  MoveL 11286 to (240.02, 46.51, 153.89) mm, rotated rx 180 ry 0 rz 180 deg; joints [-155.698, -65.543, -49.369, 46.991, 34.25, -41.545]
  MoveL 11287 to (240.02, 46.51, 153.89) mm, rotated rx 180 ry 0 rz 180 deg; joints [-155.698, -65.543, -49.369, 46.991, 34.25, -41.545]
  Call Extruder(208.81911)
  MoveL 11288 to (240.06, 46.72, 153.89) mm, rotated rx -180 ry 0 rz -180 deg; joints [-155.682, -65.561, -49.333, 47.032, 34.249, -41.586]
  MoveL 11289 to (240.06, 46.72, 153.89) mm, rotated rx -180 ry 0 rz -180 deg; joints [-155.682, -65.561, -49.333, 47.032, 34.249, -41.586]
  Call Extruder(208.93371)
  MoveL 11290 to (240.11, 46.92, 153.89) mm, rotated rx 180 ry 0 rz 180 deg; joints [-155.665, -65.578, -49.298, 47.072, 34.247, -41.627]
  MoveL 11291 to (240.11, 46.92, 153.89) mm, rotated rx 180 ry 0 rz 180 deg; joints [-155.665, -65.578, -49.298, 47.072, 34.247, -41.627]
  Call Extruder(209.04786)
  MoveL 11292 to (240.15, 47.12, 153.89) mm, rotated rx 180 ry 0 rz 180 deg; joints [-155.649, -65.596, -49.263, 47.113, 34.246, -41.668]
  MoveL 11293 to (240.15, 47.12, 153.89) mm, rotated rx 180 ry 0 rz 180 deg; joints [-155.649, -65.596, -49.263, 47.113, 34.246, -41.668]
  Call Extruder(209.16155)
  MoveL 11294 to (240.2, 47.33, 153.89) mm, rotated rx 180 ry 0 rz 180 deg; joints [-155.633, -65.614, -49.227, 47.154, 34.245, -41.71]
  MoveL 11295 to (240.2, 47.33, 153.89) mm, rotated rx 180 ry 0 rz 180 deg; joints [-155.633, -65.614, -49.227, 47.154, 34.245, -41.71]
  Call Extruder(209.28696)
  MoveL 11296 to (240.24, 47.55, 153.89) mm, rotated rx 180 ry 0 rz 180 deg; joints [-155.614, -65.633, -49.188, 47.199, 34.244, -41.755]
  MoveL 11297 to (240.24, 47.55, 153.89) mm, rotated rx 180 ry 0 rz 180 deg; joints [-155.614, -65.633, -49.188, 47.199, 34.244, -41.755]
  Call Extruder(209.42394)
  MoveL 11298 to (240.29, 47.8, 153.89) mm, rotated rx 180 ry 0 rz 180 deg; joints [-155.594, -65.654, -49.146, 47.249, 34.243, -41.804]
  MoveL 11299 to (240.29, 47.8, 153.89) mm, rotated rx 180 ry 0 rz 180 deg; joints [-155.594, -65.654, -49.146, 47.249, 34.243, -41.804]
  Call Extruder(209.56031)
  MoveL 11300 to (240.34, 48.05, 153.89) mm, rotated rx 180 ry 0 rz 180 deg; joints [-155.574, -65.675, -49.104, 47.298, 34.242, -41.854]
  MoveL 11301 to (240.34, 48.05, 153.89) mm, rotated rx 180 ry 0 rz 180 deg; joints [-155.574, -65.675, -49.104, 47.298, 34.242, -41.854]
  Call Extruder(209.69607)
  MoveL 11302 to (240.39, 48.3, 153.89) mm, rotated rx 180 ry 0 rz 180 deg; joints [-155.554, -65.696, -49.061, 47.348, 34.241, -41.904]
  MoveL 11303 to (240.39, 48.3, 153.89) mm, rotated rx 180 ry 0 rz 180 deg; joints [-155.554, -65.696, -49.061, 47.348, 34.241, -41.904]
  Call Extruder(209.83121)
  MoveL 11304 to (240.44, 48.55, 153.89) mm, rotated rx 180 ry 0 rz 180 deg; joints [-155.534, -65.717, -49.019, 47.398, 34.24, -41.954]
  MoveL 11305 to (240.44, 48.55, 153.89) mm, rotated rx 180 ry 0 rz 180 deg; joints [-155.534, -65.717, -49.019, 47.398, 34.24, -41.954]
  Call Extruder(209.96575)
  MoveL 11306 to (240.49, 48.8, 153.89) mm, rotated rx -180 ry 0 rz 180 deg; joints [-155.514, -65.738, -48.977, 47.447, 34.239, -42.003]
  MoveL 11307 to (240.49, 48.8, 153.89) mm, rotated rx -180 ry 0 rz 180 deg; joints [-155.514, -65.738, -48.977, 47.447, 34.239, -42.003]
  Call Extruder(210.09968)
  MoveL 11308 to (240.54, 49.05, 153.89) mm, rotated rx 180 ry 0 rz 180 deg; joints [-155.494, -65.759, -48.935, 47.497, 34.238, -42.053]
  MoveL 11309 to (240.54, 49.05, 153.89) mm, rotated rx 180 ry 0 rz 180 deg; joints [-155.494, -65.759, -48.935, 47.497, 34.238, -42.053]
  Call Extruder(210.24754)
  MoveL 11310 to (240.59, 49.33, 153.89) mm, rotated rx -180 ry 0 rz 180 deg; joints [-155.471, -65.782, -48.889, 47.551, 34.238, -42.108]
  MoveL 11311 to (240.59, 49.33, 153.89) mm, rotated rx -180 ry 0 rz 180 deg; joints [-155.471, -65.782, -48.889, 47.551, 34.238, -42.108]
  Call Extruder(210.40929)
  MoveL 11312 to (240.64, 49.63, 153.89) mm, rotated rx 180 ry 0 rz -180 deg; joints [-155.446, -65.806, -48.84, 47.611, 34.238, -42.167]
  MoveL 11313 to (240.64, 49.63, 153.89) mm, rotated rx 180 ry 0 rz -180 deg; joints [-155.446, -65.806, -48.84, 47.611, 34.238, -42.167]
  Call Extruder(210.57031)
  MoveL 11314 to (240.69, 49.94, 153.89) mm, rotated rx -180 ry 0 rz 180 deg; joints [-155.421, -65.831, -48.791, 47.671, 34.238, -42.227]
  MoveL 11315 to (240.69, 49.94, 153.89) mm, rotated rx -180 ry 0 rz 180 deg; joints [-155.421, -65.831, -48.791, 47.671, 34.238, -42.227]
  Call Extruder(210.73060)
  MoveL 11316 to (240.74, 50.24, 153.89) mm, rotated rx -180 ry 0 rz 180 deg; joints [-155.396, -65.855, -48.742, 47.73, 34.239, -42.287]
  MoveL 11317 to (240.74, 50.24, 153.89) mm, rotated rx -180 ry 0 rz 180 deg; joints [-155.396, -65.855, -48.742, 47.73, 34.239, -42.287]
  Call Extruder(210.89016)
  MoveL 11318 to (240.78, 50.55, 153.89) mm, rotated rx 180 ry 0 rz 180 deg; joints [-155.371, -65.88, -48.693, 47.79, 34.239, -42.346]
  MoveL 11319 to (240.78, 50.55, 153.89) mm, rotated rx 180 ry 0 rz 180 deg; joints [-155.371, -65.88, -48.693, 47.79, 34.239, -42.346]
  Call Extruder(211.04899)
  MoveL 11320 to (240.83, 50.86, 153.89) mm, rotated rx 180 ry 0 rz 180 deg; joints [-155.346, -65.904, -48.644, 47.85, 34.239, -42.406]
  MoveL 11321 to (240.83, 50.86, 153.89) mm, rotated rx 180 ry 0 rz 180 deg; joints [-155.346, -65.904, -48.644, 47.85, 34.239, -42.406]
  Call Extruder(211.22766)
  MoveL 11322 to (240.88, 51.2, 153.89) mm, rotated rx 180 ry 0 rz 180 deg; joints [-155.317, -65.931, -48.59, 47.917, 34.241, -42.473]
  MoveL 11323 to (240.88, 51.2, 153.89) mm, rotated rx 180 ry 0 rz 180 deg; joints [-155.317, -65.931, -48.59, 47.917, 34.241, -42.473]
  Call Extruder(211.42611)
  MoveL 11324 to (240.92, 51.59, 153.89) mm, rotated rx 180 ry 0 rz -180 deg; joints [-155.285, -65.96, -48.531, 47.991, 34.243, -42.546]
  MoveL 11325 to (240.92, 51.59, 153.89) mm, rotated rx 180 ry 0 rz -180 deg; joints [-155.285, -65.96, -48.531, 47.991, 34.243, -42.546]
  Call Extruder(211.62368)
  MoveL 11326 to (240.97, 51.98, 153.89) mm, rotated rx 180 ry 0 rz -180 deg; joints [-155.252, -65.989, -48.473, 48.066, 34.245, -42.62]
  MoveL 11327 to (240.97, 51.98, 153.89) mm, rotated rx 180 ry 0 rz -180 deg; joints [-155.252, -65.989, -48.473, 48.066, 34.245, -42.62]
  Call Extruder(211.82039)
  MoveL 11328 to (241.02, 52.36, 153.89) mm, rotated rx -180 ry 0 rz 180 deg; joints [-155.22, -66.019, -48.414, 48.14, 34.247, -42.694]
  MoveL 11329 to (241.02, 52.36, 153.89) mm, rotated rx -180 ry 0 rz 180 deg; joints [-155.22, -66.019, -48.414, 48.14, 34.247, -42.694]
  Call Extruder(212.01622)
  MoveL 11330 to (241.06, 52.75, 153.89) mm, rotated rx 180 ry 0 rz 180 deg; joints [-155.188, -66.048, -48.356, 48.214, 34.25, -42.768]
  MoveL 11331 to (241.06, 52.75, 153.89) mm, rotated rx 180 ry 0 rz 180 deg; joints [-155.188, -66.048, -48.356, 48.214, 34.25, -42.768]
  Call Extruder(212.31166)
  MoveL 11332 to (241.11, 53.34, 153.89) mm, rotated rx -180 ry 0 rz 180 deg; joints [-155.138, -66.09, -48.272, 48.326, 34.256, -42.877]
  MoveL 11333 to (241.11, 53.34, 153.89) mm, rotated rx -180 ry 0 rz 180 deg; joints [-155.138, -66.09, -48.272, 48.326, 34.256, -42.877]
  Call Extruder(212.60577)
  MoveL 11334 to (241.16, 53.93, 153.89) mm, rotated rx -180 ry 0 rz 180 deg; joints [-155.088, -66.131, -48.188, 48.437, 34.262, -42.987]
  MoveL 11335 to (241.16, 53.93, 153.89) mm, rotated rx -180 ry 0 rz 180 deg; joints [-155.088, -66.131, -48.188, 48.437, 34.262, -42.987]
  Call Extruder(212.89854)
  MoveL 11336 to (241.2, 54.52, 153.89) mm, rotated rx -180 ry 0 rz 180 deg; joints [-155.038, -66.173, -48.104, 48.548, 34.268, -43.096]
  MoveL 11337 to (241.2, 54.52, 153.89) mm, rotated rx -180 ry 0 rz 180 deg; joints [-155.038, -66.173, -48.104, 48.548, 34.268, -43.096]
  Call Extruder(213.47199)
  MoveL 11338 to (241.25, 55.68, 153.89) mm, rotated rx 180 ry 0 rz 180 deg; joints [-154.938, -66.25, -47.95, 48.763, 34.285, -43.307]
  MoveL 11339 to (241.25, 55.68, 153.89) mm, rotated rx 180 ry 0 rz 180 deg; joints [-154.938, -66.25, -47.95, 48.763, 34.285, -43.307]
  Call Extruder(214.18582)
  MoveL 11340 to (241.29, 57.14, 153.89) mm, rotated rx 180 ry 0 rz 180 deg; joints [-154.812, -66.345, -47.76, 49.03, 34.309, -43.568]
  Call Extruder(256.25069)
  MoveL 11341 to (241.29, 142.86, 153.89) mm, rotated rx -180 ry 0 rz 180 deg; joints [-147.778, -73.071, -34.392, 64.539, 36.196, -59.459]
  Call Extruder(256.67912)
  MoveL 11342 to (241.27, 143.73, 153.89) mm, rotated rx -180 ry 0 rz 180 deg; joints [-147.711, -73.155, -34.226, 64.698, 36.219, -59.631]
  MoveL 11343 to (241.27, 143.73, 153.89) mm, rotated rx -180 ry 0 rz 180 deg; joints [-147.711, -73.155, -34.226, 64.698, 36.219, -59.631]
  Call Extruder(257.25257)
  MoveL 11344 to (241.22, 144.9, 153.89) mm, rotated rx 180 ry 0 rz 180 deg; joints [-147.62, -73.265, -34.01, 64.907, 36.253, -59.856]
  MoveL 11345 to (241.22, 144.9, 153.89) mm, rotated rx 180 ry 0 rz 180 deg; joints [-147.62, -73.265, -34.01, 64.907, 36.253, -59.856]
  Call Extruder(257.68690)
  MoveL 11346 to (241.18, 145.77, 153.89) mm, rotated rx 180 ry 0 rz 180 deg; joints [-147.551, -73.346, -33.851, 65.062, 36.279, -60.024]
  MoveL 11347 to (241.18, 145.77, 153.89) mm, rotated rx 180 ry 0 rz 180 deg; joints [-147.551, -73.346, -33.851, 65.062, 36.279, -60.024]
  Call Extruder(257.98101)
  MoveL 11348 to (241.13, 146.36, 153.89) mm, rotated rx 180 ry 0 rz -180 deg; joints [-147.504, -73.398, -33.748, 65.165, 36.299, -60.133]
  MoveL 11349 to (241.13, 146.36, 153.89) mm, rotated rx 180 ry 0 rz -180 deg; joints [-147.504, -73.398, -33.748, 65.165, 36.299, -60.133]
  Call Extruder(258.27645)
  MoveL 11350 to (241.09, 146.95, 153.89) mm, rotated rx 180 ry 0 rz 180 deg; joints [-147.457, -73.451, -33.644, 65.267, 36.318, -60.243]
  MoveL 11351 to (241.09, 146.95, 153.89) mm, rotated rx 180 ry 0 rz 180 deg; joints [-147.457, -73.451, -33.644, 65.267, 36.318, -60.243]
  Call Extruder(258.52270)
  MoveL 11352 to (241.04, 147.44, 153.89) mm, rotated rx -180 ry 0 rz 180 deg; joints [-147.417, -73.493, -33.561, 65.351, 36.335, -60.333]
  MoveL 11353 to (241.04, 147.44, 153.89) mm, rotated rx -180 ry 0 rz 180 deg; joints [-147.417, -73.493, -33.561, 65.351, 36.335, -60.333]
  Call Extruder(258.71941)
  MoveL 11354 to (240.99, 147.83, 153.89) mm, rotated rx 180 ry 0 rz -180 deg; joints [-147.386, -73.525, -33.497, 65.416, 36.35, -60.402]
  MoveL 11355 to (240.99, 147.83, 153.89) mm, rotated rx 180 ry 0 rz -180 deg; joints [-147.386, -73.525, -33.497, 65.416, 36.35, -60.402]
  Call Extruder(258.91698)
  MoveL 11356 to (240.95, 148.22, 153.89) mm, rotated rx -180 ry 0 rz 180 deg; joints [-147.354, -73.557, -33.434, 65.481, 36.364, -60.471]
  MoveL 11357 to (240.95, 148.22, 153.89) mm, rotated rx -180 ry 0 rz 180 deg; joints [-147.354, -73.557, -33.434, 65.481, 36.364, -60.471]
  Call Extruder(259.11542)
  MoveL 11358 to (240.9, 148.6, 153.89) mm, rotated rx 180 ry 0 rz -180 deg; joints [-147.322, -73.59, -33.37, 65.546, 36.379, -60.541]
  MoveL 11359 to (240.9, 148.6, 153.89) mm, rotated rx 180 ry 0 rz -180 deg; joints [-147.322, -73.59, -33.37, 65.546, 36.379, -60.541]
  Call Extruder(259.31473)
  MoveL 11360 to (240.86, 148.99, 153.89) mm, rotated rx 180 ry 0 rz 180 deg; joints [-147.291, -73.622, -33.306, 65.611, 36.393, -60.61]
  MoveL 11361 to (240.86, 148.99, 153.89) mm, rotated rx 180 ry 0 rz 180 deg; joints [-147.291, -73.622, -33.306, 65.611, 36.393, -60.61]
  Call Extruder(259.47356)
  MoveL 11362 to (240.81, 149.3, 153.89) mm, rotated rx 180 ry 0 rz 180 deg; joints [-147.265, -73.646, -33.259, 65.661, 36.406, -60.663]
  MoveL 11363 to (240.81, 149.3, 153.89) mm, rotated rx 180 ry 0 rz 180 deg; joints [-147.265, -73.646, -33.259, 65.661, 36.406, -60.663]
  Call Extruder(259.63312)
  MoveL 11364 to (240.76, 149.6, 153.89) mm, rotated rx 180 ry 0 rz 180 deg; joints [-147.24, -73.67, -33.212, 65.71, 36.419, -60.715]
  MoveL 11365 to (240.76, 149.6, 153.89) mm, rotated rx 180 ry 0 rz 180 deg; joints [-147.24, -73.67, -33.212, 65.71, 36.419, -60.715]
  Call Extruder(259.79341)
  MoveL 11366 to (240.71, 149.91, 153.89) mm, rotated rx -180 ry 0 rz 180 deg; joints [-147.214, -73.694, -33.165, 65.76, 36.431, -60.767]
  MoveL 11367 to (240.71, 149.91, 153.89) mm, rotated rx -180 ry 0 rz 180 deg; joints [-147.214, -73.694, -33.165, 65.76, 36.431, -60.767]
  Call Extruder(259.95443)
  MoveL 11368 to (240.66, 150.21, 153.89) mm, rotated rx 180 ry 0 rz 180 deg; joints [-147.189, -73.718, -33.118, 65.809, 36.444, -60.819]
  MoveL 11369 to (240.66, 150.21, 153.89) mm, rotated rx 180 ry 0 rz 180 deg; joints [-147.189, -73.718, -33.118, 65.809, 36.444, -60.819]
  Call Extruder(260.11618)
  MoveL 11370 to (240.61, 150.52, 153.89) mm, rotated rx -180 ry 0 rz 180 deg; joints [-147.163, -73.742, -33.071, 65.859, 36.457, -60.872]
  MoveL 11371 to (240.61, 150.52, 153.89) mm, rotated rx -180 ry 0 rz 180 deg; joints [-147.163, -73.742, -33.071, 65.859, 36.457, -60.872]
  Call Extruder(260.27865)
  MoveL 11372 to (240.56, 150.83, 153.89) mm, rotated rx 180 ry 0 rz -180 deg; joints [-147.138, -73.765, -33.024, 65.908, 36.47, -60.924]
  MoveL 11373 to (240.56, 150.83, 153.89) mm, rotated rx 180 ry 0 rz -180 deg; joints [-147.138, -73.765, -33.024, 65.908, 36.47, -60.924]
  Call Extruder(260.41257)
  MoveL 11374 to (240.52, 151.07, 153.89) mm, rotated rx 180 ry 0 rz 180 deg; joints [-147.117, -73.784, -32.988, 65.947, 36.481, -60.965]
  MoveL 11375 to (240.52, 151.07, 153.89) mm, rotated rx 180 ry 0 rz 180 deg; joints [-147.117, -73.784, -32.988, 65.947, 36.481, -60.965]
  Call Extruder(260.54711)
  MoveL 11376 to (240.47, 151.32, 153.89) mm, rotated rx 180 ry 0 rz -180 deg; joints [-147.095, -73.801, -32.953, 65.986, 36.493, -61.006]
  MoveL 11377 to (240.47, 151.32, 153.89) mm, rotated rx 180 ry 0 rz -180 deg; joints [-147.095, -73.801, -32.953, 65.986, 36.493, -61.006]
  Call Extruder(260.68226)
  MoveL 11378 to (240.42, 151.57, 153.89) mm, rotated rx -180 ry 0 rz -180 deg; joints [-147.074, -73.819, -32.918, 66.025, 36.504, -61.046]
  MoveL 11379 to (240.42, 151.57, 153.89) mm, rotated rx -180 ry 0 rz -180 deg; joints [-147.074, -73.819, -32.918, 66.025, 36.504, -61.046]
  Call Extruder(260.81801)
  MoveL 11380 to (240.37, 151.82, 153.89) mm, rotated rx 180 ry 0 rz -180 deg; joints [-147.053, -73.837, -32.882, 66.064, 36.515, -61.087]
  MoveL 11381 to (240.37, 151.82, 153.89) mm, rotated rx 180 ry 0 rz -180 deg; joints [-147.053, -73.837, -32.882, 66.064, 36.515, -61.087]
  Call Extruder(260.95438)
  MoveL 11382 to (240.32, 152.07, 153.89) mm, rotated rx 180 ry 0 rz 180 deg; joints [-147.032, -73.855, -32.847, 66.102, 36.527, -61.128]
  MoveL 11383 to (240.32, 152.07, 153.89) mm, rotated rx 180 ry 0 rz 180 deg; joints [-147.032, -73.855, -32.847, 66.102, 36.527, -61.128]
  Call Extruder(261.09136)
  MoveL 11384 to (240.27, 152.32, 153.89) mm, rotated rx 180 ry 0 rz 180 deg; joints [-147.011, -73.874, -32.811, 66.141, 36.538, -61.169]
  MoveL 11385 to (240.27, 152.32, 153.89) mm, rotated rx 180 ry 0 rz 180 deg; joints [-147.011, -73.874, -32.811, 66.141, 36.538, -61.169]
  Call Extruder(261.22895)
  MoveL 11386 to (240.22, 152.57, 153.89) mm, rotated rx 180 ry 0 rz 180 deg; joints [-146.989, -73.892, -32.775, 66.18, 36.55, -61.209]
  MoveL 11387 to (240.22, 152.57, 153.89) mm, rotated rx 180 ry 0 rz 180 deg; joints [-146.989, -73.892, -32.775, 66.18, 36.55, -61.209]
  Call Extruder(261.34265)
  MoveL 11388 to (240.17, 152.77, 153.89) mm, rotated rx 180 ry 0 rz 180 deg; joints [-146.972, -73.906, -32.747, 66.211, 36.56, -61.242]
  MoveL 11389 to (240.17, 152.77, 153.89) mm, rotated rx 180 ry 0 rz 180 deg; joints [-146.972, -73.906, -32.747, 66.211, 36.56, -61.242]
  Call Extruder(261.45680)
  MoveL 11390 to (240.13, 152.98, 153.89) mm, rotated rx 180 ry 0 rz -180 deg; joints [-146.954, -73.92, -32.719, 66.242, 36.57, -61.275]
  MoveL 11391 to (240.13, 152.98, 153.89) mm, rotated rx 180 ry 0 rz -180 deg; joints [-146.954, -73.92, -32.719, 66.242, 36.57, -61.275]
  Call Extruder(261.57140)
  MoveL 11392 to (240.08, 153.18, 153.89) mm, rotated rx -180 ry 0 rz 180 deg; joints [-146.937, -73.935, -32.691, 66.274, 36.579, -61.307]
  MoveL 11393 to (240.08, 153.18, 153.89) mm, rotated rx -180 ry 0 rz 180 deg; joints [-146.937, -73.935, -32.691, 66.274, 36.579, -61.307]
  Call Extruder(261.68645)
  MoveL 11394 to (240.04, 153.39, 153.89) mm, rotated rx 180 ry 0 rz -180 deg; joints [-146.919, -73.949, -32.663, 66.305, 36.589, -61.34]
  MoveL 11395 to (240.04, 153.39, 153.89) mm, rotated rx 180 ry 0 rz -180 deg; joints [-146.919, -73.949, -32.663, 66.305, 36.589, -61.34]
  Call Extruder(261.80867)
  MoveL 11396 to (239.98, 153.6, 153.89) mm, rotated rx -180 ry 0 rz 180 deg; joints [-146.9, -73.962, -32.636, 66.336, 36.6, -61.372]
  MoveL 11397 to (239.98, 153.6, 153.89) mm, rotated rx -180 ry 0 rz 180 deg; joints [-146.9, -73.962, -32.636, 66.336, 36.6, -61.372]
  Call Extruder(261.93833)
  MoveL 11398 to (239.92, 153.82, 153.89) mm, rotated rx 180 ry 0 rz -180 deg; joints [-146.88, -73.975, -32.611, 66.367, 36.613, -61.404]
  MoveL 11399 to (239.92, 153.82, 153.89) mm, rotated rx 180 ry 0 rz -180 deg; joints [-146.88, -73.975, -32.611, 66.367, 36.613, -61.404]
  Call Extruder(262.06856)
  MoveL 11400 to (239.85, 154.05, 153.89) mm, rotated rx 180 ry 0 rz 180 deg; joints [-146.86, -73.988, -32.587, 66.399, 36.626, -61.435]
  MoveL 11401 to (239.85, 154.05, 153.89) mm, rotated rx 180 ry 0 rz 180 deg; joints [-146.86, -73.988, -32.587, 66.399, 36.626, -61.435]
  Call Extruder(262.19935)
  MoveL 11402 to (239.78, 154.27, 153.89) mm, rotated rx -180 ry 0 rz -180 deg; joints [-146.84, -74, -32.561, 66.43, 36.639, -61.467]
  MoveL 11403 to (239.78, 154.27, 153.89) mm, rotated rx -180 ry 0 rz -180 deg; joints [-146.84, -74, -32.561, 66.43, 36.639, -61.467]
  Call Extruder(262.33071)
  MoveL 11404 to (239.71, 154.49, 153.89) mm, rotated rx 180 ry 0 rz -180 deg; joints [-146.82, -74.013, -32.536, 66.461, 36.652, -61.499]
  MoveL 11405 to (239.71, 154.49, 153.89) mm, rotated rx 180 ry 0 rz -180 deg; joints [-146.82, -74.013, -32.536, 66.461, 36.652, -61.499]
  Call Extruder(262.44261)
  MoveL 11406 to (239.65, 154.68, 153.89) mm, rotated rx -180 ry 0 rz -180 deg; joints [-146.803, -74.023, -32.517, 66.487, 36.663, -61.525]
  MoveL 11407 to (239.65, 154.68, 153.89) mm, rotated rx -180 ry 0 rz -180 deg; joints [-146.803, -74.023, -32.517, 66.487, 36.663, -61.525]
  Call Extruder(262.55495)
  MoveL 11408 to (239.59, 154.87, 153.89) mm, rotated rx -180 ry 0 rz 180 deg; joints [-146.785, -74.033, -32.497, 66.513, 36.674, -61.551]
  MoveL 11409 to (239.59, 154.87, 153.89) mm, rotated rx -180 ry 0 rz 180 deg; joints [-146.785, -74.033, -32.497, 66.513, 36.674, -61.551]
  Call Extruder(262.66774)
  MoveL 11410 to (239.53, 155.06, 153.89) mm, rotated rx -180 ry 0 rz -180 deg; joints [-146.768, -74.043, -32.477, 66.538, 36.685, -61.577]
  MoveL 11411 to (239.53, 155.06, 153.89) mm, rotated rx -180 ry 0 rz -180 deg; joints [-146.768, -74.043, -32.477, 66.538, 36.685, -61.577]
  Call Extruder(262.78098)
  MoveL 11412 to (239.47, 155.25, 153.89) mm, rotated rx -180 ry 0 rz 180 deg; joints [-146.751, -74.054, -32.457, 66.564, 36.696, -61.603]
  MoveL 11413 to (239.47, 155.25, 153.89) mm, rotated rx -180 ry 0 rz 180 deg; joints [-146.751, -74.054, -32.457, 66.564, 36.696, -61.603]
  Call Extruder(262.89466)
  MoveL 11414 to (239.41, 155.44, 153.89) mm, rotated rx -180 ry 0 rz 180 deg; joints [-146.734, -74.064, -32.437, 66.59, 36.708, -61.629]
  MoveL 11415 to (239.41, 155.44, 153.89) mm, rotated rx -180 ry 0 rz 180 deg; joints [-146.734, -74.064, -32.437, 66.59, 36.708, -61.629]
  Call Extruder(263.07662)
  MoveL 11416 to (239.29, 155.73, 153.89) mm, rotated rx 180 ry 0 rz -180 deg; joints [-146.706, -74.075, -32.415, 66.626, 36.728, -61.664]
  MoveL 11417 to (239.29, 155.73, 153.89) mm, rotated rx 180 ry 0 rz -180 deg; joints [-146.706, -74.075, -32.415, 66.626, 36.728, -61.664]
  Call Extruder(263.25933)
  MoveL 11418 to (239.16, 156.02, 153.89) mm, rotated rx 180 ry 0 rz -180 deg; joints [-146.678, -74.087, -32.392, 66.661, 36.748, -61.699]
  MoveL 11419 to (239.16, 156.02, 153.89) mm, rotated rx 180 ry 0 rz -180 deg; joints [-146.678, -74.087, -32.392, 66.661, 36.748, -61.699]
  Call Extruder(263.42975)
  MoveL 11420 to (239.05, 156.29, 153.89) mm, rotated rx 180 ry 0 rz -180 deg; joints [-146.652, -74.097, -32.372, 66.694, 36.767, -61.73]
  MoveL 11421 to (239.05, 156.29, 153.89) mm, rotated rx 180 ry 0 rz -180 deg; joints [-146.652, -74.097, -32.372, 66.694, 36.767, -61.73]
  Call Extruder(263.58776)
  MoveL 11422 to (238.94, 156.54, 153.89) mm, rotated rx -180 ry 0 rz 180 deg; joints [-146.628, -74.106, -32.353, 66.724, 36.784, -61.759]
  MoveL 11423 to (238.94, 156.54, 153.89) mm, rotated rx -180 ry 0 rz 180 deg; joints [-146.628, -74.106, -32.353, 66.724, 36.784, -61.759]
  Call Extruder(263.74638)
  MoveL 11424 to (238.84, 156.79, 153.89) mm, rotated rx -180 ry 0 rz 180 deg; joints [-146.604, -74.116, -32.335, 66.754, 36.802, -61.788]
  MoveL 11425 to (238.84, 156.79, 153.89) mm, rotated rx -180 ry 0 rz 180 deg; joints [-146.604, -74.116, -32.335, 66.754, 36.802, -61.788]
  Call Extruder(263.95255)
  MoveL 11426 to (238.66, 157.09, 153.89) mm, rotated rx 180 ry 0 rz 180 deg; joints [-146.573, -74.12, -32.327, 66.784, 36.828, -61.814]
  MoveL 11427 to (238.66, 157.09, 153.89) mm, rotated rx 180 ry 0 rz 180 deg; joints [-146.573, -74.12, -32.327, 66.784, 36.828, -61.814]
  Call Extruder(264.15949)
  MoveL 11428 to (238.49, 157.4, 153.89) mm, rotated rx 180 ry 0 rz 180 deg; joints [-146.542, -74.124, -32.319, 66.813, 36.854, -61.84]
  MoveL 11429 to (238.49, 157.4, 153.89) mm, rotated rx 180 ry 0 rz 180 deg; joints [-146.542, -74.124, -32.319, 66.813, 36.854, -61.84]
  Call Extruder(264.36722)
  MoveL 11430 to (238.31, 157.7, 153.89) mm, rotated rx 180 ry 0 rz -180 deg; joints [-146.51, -74.128, -32.31, 66.843, 36.88, -61.866]
  MoveL 11431 to (238.31, 157.7, 153.89) mm, rotated rx 180 ry 0 rz -180 deg; joints [-146.51, -74.128, -32.31, 66.843, 36.88, -61.866]
  Call Extruder(264.57572)
  MoveL 11432 to (238.13, 158.01, 153.89) mm, rotated rx 180 ry 0 rz 180 deg; joints [-146.479, -74.132, -32.302, 66.873, 36.906, -61.892]
  MoveL 11433 to (238.13, 158.01, 153.89) mm, rotated rx 180 ry 0 rz 180 deg; joints [-146.479, -74.132, -32.302, 66.873, 36.906, -61.892]
  Call Extruder(264.75269)
  MoveL 11434 to (237.96, 158.25, 153.89) mm, rotated rx 180 ry 0 rz 180 deg; joints [-146.452, -74.13, -32.307, 66.891, 36.93, -61.905]
  MoveL 11435 to (237.96, 158.25, 153.89) mm, rotated rx 180 ry 0 rz 180 deg; joints [-146.452, -74.13, -32.307, 66.891, 36.93, -61.905]
  Call Extruder(265.08090)
  MoveL 11436 to (237.64, 158.69, 153.89) mm, rotated rx 180 ry 0 rz 180 deg; joints [-146.403, -74.125, -32.315, 66.924, 36.976, -61.93]
  MoveL 11437 to (237.64, 158.69, 153.89) mm, rotated rx 180 ry 0 rz 180 deg; joints [-146.403, -74.125, -32.315, 66.924, 36.976, -61.93]
  Call Extruder(265.41030)
  MoveL 11438 to (237.32, 159.14, 153.89) mm, rotated rx -180 ry 0 rz -180 deg; joints [-146.354, -74.121, -32.324, 66.957, 37.021, -61.954]
  Call Extruder(266.28192)
  MoveL 11439 to (236.35, 160.23, 153.89) mm, rotated rx 180 ry 0 rz -180 deg; joints [-146.225, -74.083, -32.399, 67.013, 37.149, -61.978]
  Call Extruder(267.07895)
  MoveL 11440 to (235.35, 161.1, 153.89) mm, rotated rx -180 ry 0 rz 180 deg; joints [-146.109, -74.017, -32.53, 67.025, 37.276, -61.951]
  Call Extruder(267.24365)
  MoveL 11441 to (235.13, 161.26, 153.89) mm, rotated rx 180 ry 0 rz 180 deg; joints [-146.086, -73.998, -32.566, 67.022, 37.303, -61.939]
  MoveL 11442 to (235.13, 161.26, 153.89) mm, rotated rx 180 ry 0 rz 180 deg; joints [-146.086, -73.998, -32.566, 67.022, 37.303, -61.939]
  Call Extruder(267.57190)
  MoveL 11443 to (234.69, 161.59, 153.89) mm, rotated rx 180 ry 0 rz -180 deg; joints [-146.04, -73.962, -32.638, 67.015, 37.358, -61.914]
  MoveL 11444 to (234.69, 161.59, 153.89) mm, rotated rx 180 ry 0 rz -180 deg; joints [-146.04, -73.962, -32.638, 67.015, 37.358, -61.914]
  Call Extruder(267.89900)
  MoveL 11445 to (234.24, 161.91, 153.89) mm, rotated rx 180 ry 0 rz 180 deg; joints [-145.993, -73.926, -32.709, 67.009, 37.413, -61.889]
  MoveL 11446 to (234.24, 161.91, 153.89) mm, rotated rx 180 ry 0 rz 180 deg; joints [-145.993, -73.926, -32.709, 67.009, 37.413, -61.889]
  Call Extruder(268.03352)
  MoveL 11447 to (234.05, 162.03, 153.89) mm, rotated rx 180 ry 0 rz 180 deg; joints [-145.975, -73.906, -32.746, 67.001, 37.436, -61.873]
  MoveL 11448 to (234.05, 162.03, 153.89) mm, rotated rx 180 ry 0 rz 180 deg; joints [-145.975, -73.906, -32.746, 67.001, 37.436, -61.873]
  Call Extruder(268.24883)
  MoveL 11449 to (233.73, 162.21, 153.89) mm, rotated rx 180 ry 0 rz 180 deg; joints [-145.946, -73.876, -32.807, 66.987, 37.474, -61.845]
  MoveL 11450 to (233.73, 162.21, 153.89) mm, rotated rx 180 ry 0 rz 180 deg; joints [-145.946, -73.876, -32.807, 66.987, 37.474, -61.845]
  Call Extruder(268.46330)
  MoveL 11451 to (233.42, 162.39, 153.89) mm, rotated rx -180 ry 0 rz 180 deg; joints [-145.916, -73.845, -32.868, 66.974, 37.511, -61.818]
  MoveL 11452 to (233.42, 162.39, 153.89) mm, rotated rx -180 ry 0 rz 180 deg; joints [-145.916, -73.845, -32.868, 66.974, 37.511, -61.818]
  Call Extruder(268.67694)
  MoveL 11453 to (233.1, 162.57, 153.89) mm, rotated rx 180 ry 0 rz 180 deg; joints [-145.887, -73.814, -32.928, 66.961, 37.549, -61.791]
  MoveL 11454 to (233.1, 162.57, 153.89) mm, rotated rx 180 ry 0 rz 180 deg; joints [-145.887, -73.814, -32.928, 66.961, 37.549, -61.791]
  Call Extruder(268.85614)
  MoveL 11455 to (232.83, 162.71, 153.89) mm, rotated rx -180 ry 0 rz 180 deg; joints [-145.863, -73.786, -32.984, 66.947, 37.581, -61.765]
  MoveL 11456 to (232.83, 162.71, 153.89) mm, rotated rx -180 ry 0 rz 180 deg; joints [-145.863, -73.786, -32.984, 66.947, 37.581, -61.765]
  Call Extruder(269.00184)
  MoveL 11457 to (232.6, 162.81, 153.89) mm, rotated rx 180 ry 0 rz 180 deg; joints [-145.844, -73.76, -33.035, 66.932, 37.607, -61.739]
  MoveL 11458 to (232.6, 162.81, 153.89) mm, rotated rx 180 ry 0 rz 180 deg; joints [-145.844, -73.76, -33.035, 66.932, 37.607, -61.739]
  Call Extruder(269.14703)
  MoveL 11459 to (232.37, 162.91, 153.89) mm, rotated rx 180 ry 0 rz 180 deg; joints [-145.825, -73.734, -33.086, 66.917, 37.634, -61.713]
  MoveL 11460 to (232.37, 162.91, 153.89) mm, rotated rx 180 ry 0 rz 180 deg; joints [-145.825, -73.734, -33.086, 66.917, 37.634, -61.713]
  Call Extruder(269.32977)
  MoveL 11461 to (232.07, 163.02, 153.89) mm, rotated rx 180 ry 0 rz 180 deg; joints [-145.801, -73.701, -33.152, 66.897, 37.667, -61.678]
  MoveL 11462 to (232.07, 163.02, 153.89) mm, rotated rx 180 ry 0 rz 180 deg; joints [-145.801, -73.701, -33.152, 66.897, 37.667, -61.678]
  Call Extruder(269.51175)
  MoveL 11463 to (231.78, 163.15, 153.89) mm, rotated rx -180 ry 0 rz -180 deg; joints [-145.777, -73.668, -33.217, 66.877, 37.701, -61.645]
  MoveL 11464 to (231.78, 163.15, 153.89) mm, rotated rx -180 ry 0 rz -180 deg; joints [-145.777, -73.668, -33.217, 66.877, 37.701, -61.645]
  Call Extruder(269.65909)
  MoveL 11465 to (231.54, 163.24, 153.89) mm, rotated rx -180 ry 0 rz -180 deg; joints [-145.759, -73.639, -33.272, 66.859, 37.728, -61.615]
  MoveL 11466 to (231.54, 163.24, 153.89) mm, rotated rx -180 ry 0 rz -180 deg; joints [-145.759, -73.639, -33.272, 66.859, 37.728, -61.615]
  Call Extruder(269.77231)
  MoveL 11467 to (231.35, 163.3, 153.89) mm, rotated rx 180 ry 0 rz 180 deg; joints [-145.744, -73.616, -33.318, 66.844, 37.749, -61.591]
  MoveL 11468 to (231.35, 163.3, 153.89) mm, rotated rx 180 ry 0 rz 180 deg; joints [-145.744, -73.616, -33.318, 66.844, 37.749, -61.591]
  Call Extruder(269.88509)
  MoveL 11469 to (231.17, 163.36, 153.89) mm, rotated rx -180 ry 0 rz 180 deg; joints [-145.73, -73.593, -33.363, 66.828, 37.77, -61.566]
  MoveL 11470 to (231.17, 163.36, 153.89) mm, rotated rx -180 ry 0 rz 180 deg; joints [-145.73, -73.593, -33.363, 66.828, 37.77, -61.566]
  Call Extruder(269.99742)
  MoveL 11471 to (230.98, 163.42, 153.89) mm, rotated rx 180 ry 0 rz -180 deg; joints [-145.716, -73.57, -33.409, 66.812, 37.792, -61.541]
  MoveL 11472 to (230.98, 163.42, 153.89) mm, rotated rx 180 ry 0 rz -180 deg; joints [-145.716, -73.57, -33.409, 66.812, 37.792, -61.541]
  Call Extruder(270.10931)
  MoveL 11473 to (230.79, 163.48, 153.89) mm, rotated rx 180 ry 0 rz -180 deg; joints [-145.702, -73.547, -33.454, 66.797, 37.813, -61.516]
  MoveL 11474 to (230.79, 163.48, 153.89) mm, rotated rx 180 ry 0 rz -180 deg; joints [-145.702, -73.547, -33.454, 66.797, 37.813, -61.516]
  Call Extruder(270.23072)
  MoveL 11475 to (230.58, 163.55, 153.89) mm, rotated rx 180 ry 0 rz 180 deg; joints [-145.687, -73.522, -33.504, 66.78, 37.836, -61.488]
  MoveL 11476 to (230.58, 163.55, 153.89) mm, rotated rx 180 ry 0 rz 180 deg; joints [-145.687, -73.522, -33.504, 66.78, 37.836, -61.488]
  Call Extruder(270.36153)
  MoveL 11477 to (230.36, 163.61, 153.89) mm, rotated rx 180 ry 0 rz 180 deg; joints [-145.67, -73.494, -33.559, 66.761, 37.861, -61.458]
  MoveL 11478 to (230.36, 163.61, 153.89) mm, rotated rx 180 ry 0 rz 180 deg; joints [-145.67, -73.494, -33.559, 66.761, 37.861, -61.458]
  Call Extruder(270.49178)
  MoveL 11479 to (230.14, 163.68, 153.89) mm, rotated rx -180 ry 0 rz 180 deg; joints [-145.654, -73.466, -33.613, 66.742, 37.886, -61.428]
  MoveL 11480 to (230.14, 163.68, 153.89) mm, rotated rx -180 ry 0 rz 180 deg; joints [-145.654, -73.466, -33.613, 66.742, 37.886, -61.428]
  Call Extruder(270.62146)
  MoveL 11481 to (229.91, 163.75, 153.89) mm, rotated rx -180 ry 0 rz 180 deg; joints [-145.638, -73.439, -33.668, 66.723, 37.911, -61.398]
  MoveL 11482 to (229.91, 163.75, 153.89) mm, rotated rx -180 ry 0 rz 180 deg; joints [-145.638, -73.439, -33.668, 66.723, 37.911, -61.398]
  Call Extruder(270.75058)
  MoveL 11483 to (229.69, 163.82, 153.89) mm, rotated rx 180 ry 0 rz 180 deg; joints [-145.621, -73.411, -33.723, 66.704, 37.936, -61.368]
  MoveL 11484 to (229.69, 163.82, 153.89) mm, rotated rx 180 ry 0 rz 180 deg; joints [-145.621, -73.411, -33.723, 66.704, 37.936, -61.368]
  Call Extruder(270.86565)
  MoveL 11485 to (229.48, 163.86, 153.89) mm, rotated rx 180 ry 0 rz 180 deg; joints [-145.607, -73.384, -33.776, 66.684, 37.959, -61.337]
  MoveL 11486 to (229.48, 163.86, 153.89) mm, rotated rx 180 ry 0 rz 180 deg; joints [-145.607, -73.384, -33.776, 66.684, 37.959, -61.337]
  Call Extruder(270.98027)
  MoveL 11487 to (229.28, 163.91, 153.89) mm, rotated rx 180 ry 0 rz -180 deg; joints [-145.594, -73.357, -33.829, 66.664, 37.981, -61.306]
  MoveL 11488 to (229.28, 163.91, 153.89) mm, rotated rx 180 ry 0 rz -180 deg; joints [-145.594, -73.357, -33.829, 66.664, 37.981, -61.306]
  Call Extruder(271.09444)
  MoveL 11489 to (229.08, 163.95, 153.89) mm, rotated rx 180 ry 0 rz -180 deg; joints [-145.58, -73.33, -33.882, 66.643, 38.003, -61.276]
  MoveL 11490 to (229.08, 163.95, 153.89) mm, rotated rx 180 ry 0 rz -180 deg; joints [-145.58, -73.33, -33.882, 66.643, 38.003, -61.276]
  Call Extruder(271.20816)
  MoveL 11491 to (228.87, 164, 153.89) mm, rotated rx -180 ry 0 rz -180 deg; joints [-145.566, -73.303, -33.935, 66.623, 38.026, -61.245]
  MoveL 11492 to (228.87, 164, 153.89) mm, rotated rx -180 ry 0 rz -180 deg; joints [-145.566, -73.303, -33.935, 66.623, 38.026, -61.245]
  Call Extruder(271.33358)
  MoveL 11493 to (228.65, 164.04, 153.89) mm, rotated rx 180 ry 0 rz 180 deg; joints [-145.551, -73.273, -33.995, 66.601, 38.051, -61.211]
  MoveL 11494 to (228.65, 164.04, 153.89) mm, rotated rx 180 ry 0 rz 180 deg; joints [-145.551, -73.273, -33.995, 66.601, 38.051, -61.211]
  Call Extruder(271.47056)
  MoveL 11495 to (228.4, 164.09, 153.89) mm, rotated rx 180 ry 0 rz 180 deg; joints [-145.535, -73.24, -34.06, 66.576, 38.078, -61.173]
  MoveL 11496 to (228.4, 164.09, 153.89) mm, rotated rx 180 ry 0 rz 180 deg; joints [-145.535, -73.24, -34.06, 66.576, 38.078, -61.173]
  Call Extruder(271.60692)
  MoveL 11497 to (228.15, 164.14, 153.89) mm, rotated rx 180 ry 0 rz 180 deg; joints [-145.518, -73.206, -34.126, 66.551, 38.105, -61.135]
  MoveL 11498 to (228.15, 164.14, 153.89) mm, rotated rx 180 ry 0 rz 180 deg; joints [-145.518, -73.206, -34.126, 66.551, 38.105, -61.135]
  Call Extruder(271.74268)
  MoveL 11499 to (227.9, 164.19, 153.89) mm, rotated rx 180 ry 0 rz 180 deg; joints [-145.502, -73.173, -34.191, 66.526, 38.132, -61.097]
  MoveL 11500 to (227.9, 164.19, 153.89) mm, rotated rx 180 ry 0 rz 180 deg; joints [-145.502, -73.173, -34.191, 66.526, 38.132, -61.097]
  Call Extruder(271.87783)
  MoveL 11501 to (227.65, 164.24, 153.89) mm, rotated rx -180 ry 0 rz 180 deg; joints [-145.485, -73.14, -34.256, 66.502, 38.16, -61.06]
  MoveL 11502 to (227.65, 164.24, 153.89) mm, rotated rx -180 ry 0 rz 180 deg; joints [-145.485, -73.14, -34.256, 66.502, 38.16, -61.06]
  Call Extruder(272.01237)
  MoveL 11503 to (227.4, 164.29, 153.89) mm, rotated rx 180 ry 0 rz 180 deg; joints [-145.469, -73.107, -34.321, 66.477, 38.187, -61.022]
  MoveL 11504 to (227.4, 164.29, 153.89) mm, rotated rx 180 ry 0 rz 180 deg; joints [-145.469, -73.107, -34.321, 66.477, 38.187, -61.022]
  Call Extruder(272.14629)
  MoveL 11505 to (227.15, 164.34, 153.89) mm, rotated rx 180 ry 0 rz 180 deg; joints [-145.453, -73.074, -34.387, 66.453, 38.214, -60.985]
  MoveL 11506 to (227.15, 164.34, 153.89) mm, rotated rx 180 ry 0 rz 180 deg; joints [-145.453, -73.074, -34.387, 66.453, 38.214, -60.985]
  Call Extruder(272.29416)
  MoveL 11507 to (226.87, 164.39, 153.89) mm, rotated rx -180 ry 0 rz -180 deg; joints [-145.435, -73.037, -34.46, 66.424, 38.244, -60.942]
  MoveL 11508 to (226.87, 164.39, 153.89) mm, rotated rx -180 ry 0 rz -180 deg; joints [-145.435, -73.037, -34.46, 66.424, 38.244, -60.942]
  Call Extruder(272.45590)
  MoveL 11509 to (226.57, 164.44, 153.89) mm, rotated rx 180 ry 0 rz -180 deg; joints [-145.415, -72.995, -34.542, 66.393, 38.277, -60.894]
  MoveL 11510 to (226.57, 164.44, 153.89) mm, rotated rx 180 ry 0 rz -180 deg; joints [-145.415, -72.995, -34.542, 66.393, 38.277, -60.894]
  Call Extruder(272.61691)
  MoveL 11511 to (226.26, 164.49, 153.89) mm, rotated rx 180 ry 0 rz 180 deg; joints [-145.396, -72.953, -34.624, 66.361, 38.31, -60.846]
  MoveL 11512 to (226.26, 164.49, 153.89) mm, rotated rx 180 ry 0 rz 180 deg; joints [-145.396, -72.953, -34.624, 66.361, 38.31, -60.846]
  Call Extruder(272.77720)
  MoveL 11513 to (225.96, 164.53, 153.89) mm, rotated rx -180 ry 0 rz 180 deg; joints [-145.377, -72.912, -34.706, 66.329, 38.343, -60.799]
  MoveL 11514 to (225.96, 164.53, 153.89) mm, rotated rx -180 ry 0 rz 180 deg; joints [-145.377, -72.912, -34.706, 66.329, 38.343, -60.799]
  Call Extruder(272.93675)
  MoveL 11515 to (225.65, 164.58, 153.89) mm, rotated rx -180 ry 0 rz -180 deg; joints [-145.357, -72.871, -34.788, 66.298, 38.376, -60.751]
  MoveL 11516 to (225.65, 164.58, 153.89) mm, rotated rx -180 ry 0 rz -180 deg; joints [-145.357, -72.871, -34.788, 66.298, 38.376, -60.751]
  Call Extruder(273.09558)
  MoveL 11517 to (225.34, 164.63, 153.89) mm, rotated rx -180 ry 0 rz 180 deg; joints [-145.338, -72.829, -34.869, 66.267, 38.409, -60.704]
  MoveL 11518 to (225.34, 164.63, 153.89) mm, rotated rx -180 ry 0 rz 180 deg; joints [-145.338, -72.829, -34.869, 66.267, 38.409, -60.704]
  Call Extruder(273.27425)
  MoveL 11519 to (225, 164.68, 153.89) mm, rotated rx -180 ry 0 rz 180 deg; joints [-145.317, -72.782, -34.963, 66.23, 38.447, -60.649]
  MoveL 11520 to (225, 164.68, 153.89) mm, rotated rx -180 ry 0 rz 180 deg; joints [-145.317, -72.782, -34.963, 66.23, 38.447, -60.649]
  Call Extruder(273.47269)
  MoveL 11521 to (224.61, 164.72, 153.89) mm, rotated rx -180 ry 0 rz 180 deg; joints [-145.293, -72.728, -35.069, 66.189, 38.488, -60.587]
  MoveL 11522 to (224.61, 164.72, 153.89) mm, rotated rx -180 ry 0 rz 180 deg; joints [-145.293, -72.728, -35.069, 66.189, 38.488, -60.587]
  Call Extruder(273.67027)
  MoveL 11523 to (224.22, 164.77, 153.89) mm, rotated rx -180 ry 0 rz 180 deg; joints [-145.27, -72.674, -35.175, 66.147, 38.53, -60.524]
  MoveL 11524 to (224.22, 164.77, 153.89) mm, rotated rx -180 ry 0 rz 180 deg; joints [-145.27, -72.674, -35.175, 66.147, 38.53, -60.524]
  Call Extruder(273.86697)
  MoveL 11525 to (223.83, 164.82, 153.89) mm, rotated rx -180 ry 0 rz 180 deg; joints [-145.246, -72.621, -35.28, 66.106, 38.571, -60.463]
  MoveL 11526 to (223.83, 164.82, 153.89) mm, rotated rx -180 ry 0 rz 180 deg; joints [-145.246, -72.621, -35.28, 66.106, 38.571, -60.463]
  Call Extruder(274.06281)
  MoveL 11527 to (223.45, 164.86, 153.89) mm, rotated rx 180 ry 0 rz 180 deg; joints [-145.223, -72.568, -35.386, 66.065, 38.613, -60.401]
  MoveL 11528 to (223.45, 164.86, 153.89) mm, rotated rx 180 ry 0 rz 180 deg; joints [-145.223, -72.568, -35.386, 66.065, 38.613, -60.401]
  Call Extruder(274.35817)
  MoveL 11529 to (222.86, 164.91, 153.89) mm, rotated rx -180 ry 0 rz 180 deg; joints [-145.189, -72.484, -35.55, 65.999, 38.675, -60.303]
  MoveL 11530 to (222.86, 164.91, 153.89) mm, rotated rx -180 ry 0 rz 180 deg; joints [-145.189, -72.484, -35.55, 65.999, 38.675, -60.303]
  Call Extruder(274.65220)
  MoveL 11531 to (222.27, 164.96, 153.89) mm, rotated rx 180 ry 0 rz 180 deg; joints [-145.155, -72.401, -35.713, 65.934, 38.738, -60.206]
  MoveL 11532 to (222.27, 164.96, 153.89) mm, rotated rx 180 ry 0 rz 180 deg; joints [-145.155, -72.401, -35.713, 65.934, 38.738, -60.206]
  Call Extruder(274.94489)
  MoveL 11533 to (221.68, 165, 153.89) mm, rotated rx 180 ry 0 rz 180 deg; joints [-145.121, -72.319, -35.876, 65.87, 38.8, -60.11]
  MoveL 11534 to (221.68, 165, 153.89) mm, rotated rx 180 ry 0 rz 180 deg; joints [-145.121, -72.319, -35.876, 65.87, 38.8, -60.11]
  Call Extruder(275.51834)
  MoveL 11535 to (220.52, 165.05, 153.89) mm, rotated rx -180 ry 0 rz 180 deg; joints [-145.056, -72.152, -36.206, 65.737, 38.922, -59.914]
  MoveL 11536 to (220.52, 165.05, 153.89) mm, rotated rx -180 ry 0 rz 180 deg; joints [-145.056, -72.152, -36.206, 65.737, 38.922, -59.914]
  Call Extruder(276.23235)
  MoveL 11537 to (219.06, 165.09, 153.89) mm, rotated rx -180 ry 0 rz 180 deg; joints [-144.977, -71.944, -36.618, 65.571, 39.075, -59.668]
  Call Extruder(393.07903)
  MoveL 11538 to (-19.06, 165.09, 153.89) mm, rotated rx 180 ry 0 rz 180 deg; joints [-127.435, -50.468, -80.487, 63.354, 62.673, -42.456]
  Call Extruder(393.50763)
  MoveL 11539 to (-19.94, 165.07, 153.89) mm, rotated rx -180 ry 0 rz 180 deg; joints [-127.348, -50.417, -80.596, 63.399, 62.757, -42.43]
  MoveL 11540 to (-19.94, 165.07, 153.89) mm, rotated rx -180 ry 0 rz 180 deg; joints [-127.348, -50.417, -80.596, 63.399, 62.757, -42.43]
  Call Extruder(394.08108)
  MoveL 11541 to (-21.1, 165.03, 153.89) mm, rotated rx -180 ry 0 rz -180 deg; joints [-127.235, -50.348, -80.744, 63.457, 62.869, -42.394]
  MoveL 11542 to (-21.1, 165.03, 153.89) mm, rotated rx -180 ry 0 rz -180 deg; joints [-127.235, -50.348, -80.744, 63.457, 62.869, -42.394]
  Call Extruder(394.51538)
  MoveL 11543 to (-21.97, 164.98, 153.89) mm, rotated rx 180 ry 0 rz 180 deg; joints [-127.15, -50.295, -80.857, 63.5, 62.953, -42.365]
  MoveL 11544 to (-21.97, 164.98, 153.89) mm, rotated rx 180 ry 0 rz 180 deg; joints [-127.15, -50.295, -80.857, 63.5, 62.953, -42.365]
  Call Extruder(394.80941)
  MoveL 11545 to (-22.56, 164.93, 153.89) mm, rotated rx -180 ry 0 rz 180 deg; joints [-127.093, -50.259, -80.935, 63.527, 63.01, -42.344]
  MoveL 11546 to (-22.56, 164.93, 153.89) mm, rotated rx -180 ry 0 rz 180 deg; joints [-127.093, -50.259, -80.935, 63.527, 63.01, -42.344]
  Call Extruder(395.10477)
  MoveL 11547 to (-23.15, 164.89, 153.89) mm, rotated rx 180 ry 0 rz 180 deg; joints [-127.037, -50.222, -81.014, 63.555, 63.066, -42.324]
  MoveL 11548 to (-23.15, 164.89, 153.89) mm, rotated rx 180 ry 0 rz 180 deg; joints [-127.037, -50.222, -81.014, 63.555, 63.066, -42.324]
  Call Extruder(395.35098)
  MoveL 11549 to (-23.64, 164.84, 153.89) mm, rotated rx 180 ry 0 rz 180 deg; joints [-126.991, -50.191, -81.079, 63.577, 63.113, -42.306]
  MoveL 11550 to (-23.64, 164.84, 153.89) mm, rotated rx 180 ry 0 rz 180 deg; joints [-126.991, -50.191, -81.079, 63.577, 63.113, -42.306]
  Call Extruder(395.54769)
  MoveL 11551 to (-24.03, 164.79, 153.89) mm, rotated rx -180 ry 0 rz 180 deg; joints [-126.955, -50.166, -81.133, 63.594, 63.15, -42.29]
  MoveL 11552 to (-24.03, 164.79, 153.89) mm, rotated rx -180 ry 0 rz 180 deg; joints [-126.955, -50.166, -81.133, 63.594, 63.15, -42.29]
  Call Extruder(395.74526)
  MoveL 11553 to (-24.42, 164.75, 153.89) mm, rotated rx -180 ry 0 rz 180 deg; joints [-126.919, -50.141, -81.187, 63.611, 63.187, -42.275]
  MoveL 11554 to (-24.42, 164.75, 153.89) mm, rotated rx -180 ry 0 rz 180 deg; joints [-126.919, -50.141, -81.187, 63.611, 63.187, -42.275]
  Call Extruder(395.94370)
  MoveL 11555 to (-24.8, 164.7, 153.89) mm, rotated rx 180 ry 0 rz 180 deg; joints [-126.883, -50.116, -81.24, 63.628, 63.224, -42.26]
  MoveL 11556 to (-24.8, 164.7, 153.89) mm, rotated rx 180 ry 0 rz 180 deg; joints [-126.883, -50.116, -81.24, 63.628, 63.224, -42.26]
  Call Extruder(396.14301)
  MoveL 11557 to (-25.19, 164.66, 153.89) mm, rotated rx -180 ry 0 rz -180 deg; joints [-126.847, -50.091, -81.294, 63.645, 63.261, -42.244]
  MoveL 11558 to (-25.19, 164.66, 153.89) mm, rotated rx -180 ry 0 rz -180 deg; joints [-126.847, -50.091, -81.294, 63.645, 63.261, -42.244]
  Call Extruder(396.30184)
  MoveL 11559 to (-25.5, 164.61, 153.89) mm, rotated rx -180 ry 0 rz 180 deg; joints [-126.82, -50.071, -81.338, 63.657, 63.29, -42.231]
  MoveL 11560 to (-25.5, 164.61, 153.89) mm, rotated rx -180 ry 0 rz 180 deg; joints [-126.82, -50.071, -81.338, 63.657, 63.29, -42.231]
  Call Extruder(396.46140)
  MoveL 11561 to (-25.8, 164.56, 153.89) mm, rotated rx -180 ry 0 rz -180 deg; joints [-126.792, -50.05, -81.382, 63.669, 63.319, -42.218]
  MoveL 11562 to (-25.8, 164.56, 153.89) mm, rotated rx -180 ry 0 rz -180 deg; joints [-126.792, -50.05, -81.382, 63.669, 63.319, -42.218]
  Call Extruder(396.62169)
  MoveL 11563 to (-26.11, 164.51, 153.89) mm, rotated rx -180 ry 0 rz 180 deg; joints [-126.765, -50.03, -81.426, 63.681, 63.347, -42.204]
  MoveL 11564 to (-26.11, 164.51, 153.89) mm, rotated rx -180 ry 0 rz 180 deg; joints [-126.765, -50.03, -81.426, 63.681, 63.347, -42.204]
  Call Extruder(396.78271)
  MoveL 11565 to (-26.41, 164.46, 153.89) mm, rotated rx 180 ry 0 rz 180 deg; joints [-126.737, -50.009, -81.47, 63.693, 63.376, -42.191]
  MoveL 11566 to (-26.41, 164.46, 153.89) mm, rotated rx 180 ry 0 rz 180 deg; joints [-126.737, -50.009, -81.47, 63.693, 63.376, -42.191]
  Call Extruder(396.94445)
  MoveL 11567 to (-26.72, 164.41, 153.89) mm, rotated rx 180 ry 0 rz 180 deg; joints [-126.71, -49.989, -81.514, 63.706, 63.405, -42.178]
  MoveL 11568 to (-26.72, 164.41, 153.89) mm, rotated rx 180 ry 0 rz 180 deg; joints [-126.71, -49.989, -81.514, 63.706, 63.405, -42.178]
  Call Extruder(397.10692)
  MoveL 11569 to (-27.03, 164.36, 153.89) mm, rotated rx -180 ry 0 rz -180 deg; joints [-126.682, -49.968, -81.558, 63.718, 63.434, -42.164]
  MoveL 11570 to (-27.03, 164.36, 153.89) mm, rotated rx -180 ry 0 rz -180 deg; joints [-126.682, -49.968, -81.558, 63.718, 63.434, -42.164]
  Call Extruder(397.24085)
  MoveL 11571 to (-27.27, 164.32, 153.89) mm, rotated rx -180 ry 0 rz -180 deg; joints [-126.66, -49.951, -81.596, 63.727, 63.458, -42.152]
  MoveL 11572 to (-27.27, 164.32, 153.89) mm, rotated rx -180 ry 0 rz -180 deg; joints [-126.66, -49.951, -81.596, 63.727, 63.458, -42.152]
  Call Extruder(397.37538)
  MoveL 11573 to (-27.52, 164.27, 153.89) mm, rotated rx 180 ry 0 rz -180 deg; joints [-126.638, -49.933, -81.633, 63.736, 63.481, -42.14]
  MoveL 11574 to (-27.52, 164.27, 153.89) mm, rotated rx 180 ry 0 rz -180 deg; joints [-126.638, -49.933, -81.633, 63.736, 63.481, -42.14]
  Call Extruder(397.51053)
  MoveL 11575 to (-27.77, 164.22, 153.89) mm, rotated rx 180 ry 0 rz 180 deg; joints [-126.617, -49.916, -81.67, 63.745, 63.505, -42.128]
  MoveL 11576 to (-27.77, 164.22, 153.89) mm, rotated rx 180 ry 0 rz 180 deg; joints [-126.617, -49.916, -81.67, 63.745, 63.505, -42.128]
  Call Extruder(397.64629)
  MoveL 11577 to (-28.02, 164.17, 153.89) mm, rotated rx 180 ry 0 rz 180 deg; joints [-126.595, -49.899, -81.708, 63.755, 63.528, -42.117]
  MoveL 11578 to (-28.02, 164.17, 153.89) mm, rotated rx 180 ry 0 rz 180 deg; joints [-126.595, -49.899, -81.708, 63.755, 63.528, -42.117]
  Call Extruder(397.78265)
  MoveL 11579 to (-28.27, 164.12, 153.89) mm, rotated rx -180 ry 0 rz 180 deg; joints [-126.573, -49.881, -81.745, 63.764, 63.552, -42.105]
  MoveL 11580 to (-28.27, 164.12, 153.89) mm, rotated rx -180 ry 0 rz 180 deg; joints [-126.573, -49.881, -81.745, 63.764, 63.552, -42.105]
  Call Extruder(397.86751)
  MoveL 11581 to (-28.43, 164.09, 153.89) mm, rotated rx 180 ry 0 rz 180 deg; joints [-126.559, -49.871, -81.768, 63.77, 63.566, -42.097]
  Set speed (130.0 mm/s)
  MoveL 11582 to (-31.76, 163.31, 153.89) mm, rotated rx 180 ry 0 rz 180 deg; joints [-126.274, -49.631, -82.283, 63.884, 63.879, -41.926]
  Call Extruder(395.86751)
  Set speed (40.0 mm/s)
  MoveL 11583 to (-31.76, 163.31, 153.89) mm, rotated rx 180 ry 0 rz 180 deg; joints [-126.274, -49.631, -82.283, 63.884, 63.879, -41.926]
  Set speed (1000.0 mm/s)
  Call Extruder(-1)
  MoveL 11584 to (-31.76, 163.31, 153.89) mm, rotated rx 180 ry 0 rz 180 deg; joints [-126.274, -49.631, -82.283, 63.884, 63.879, -41.926]
  Call Extruder(0.00000)
  Call M_RunCode(107)
  Call M_RunCode(104)
  Call M_RunCode(84)
  Call M_RunCode(140)

--- Python program Extruder ---
# This macro allows simulating a 3D printing extruder
# The macro will output spray gun statistics
#
# More information about the RoboDK API here:
# https://robodk.com/doc/en/RoboDK-API.html
# For more information visit:
# http://www.robodk.com/doc/en/PythonAPI/robolink.html
#
# Define the default action (0 to deactivate, +1 to activate, -1 to clear any spray gun simulation)
# Setting it to None will display a message
ACTION = None
# Check if we are running this program inside another program and passing arguments
import sys
if len(sys.argv) > 1:
    ACTION = float(sys.argv[1])
    # For faster speed: igone values greater than 0
    if ACTION > 0:
        quit()

from robolink import *    # API to communicate with RoboDK
from robodk import *      # basic matrix operations
RDK = Robolink()

# quit if we are not in simulation mode
if RDK.RunMode() != RUNMODE_SIMULATE:
    quit()

# Get any previously added spray gun simulations and display statistics (spray on the part vs spray falling out of the part)
existing_material_simulation = False
info, stats_data = RDK.Spray_GetStats()
if stats_data.size(1) > 0:
    print("Spray gun statistics:")
    print(info)
    print(stats_data.tr())
    existing_material_simulation = True
    # # Diplay statistics
    # RDK.ShowMessage("Material used: %.1f%%<br>Material waisted: %.1f%%<br>Total particles: %.1f" % (data[1,0],data[2,0],data[3,0]), True)
    # # Clear previous spray
    # RDK.Spray_Clear()

# If the default ACTION is None, display a message to activate/deactivate the spray gun
if ACTION is None:
    print('Note: This macro can be called as Extruder(0) to turn it ON or Extruder(-1) to turn it OFF')
    entry = mbox('Turn Extruder ON or OFF', ('On', '0'), ('Off', '-1'))
    if not entry:
        quit()
    ACTION = int(entry)

if ACTION < 0:
    # Turn material deposition off
    # Select Escape to delete existing material simulations
    #RDK.Spray_Clear()
    RDK.Spray_SetState(SPRAY_OFF)

elif ACTION >= 0:

    if existing_material_simulation:
        # Select Esc key to delete existing material simulations and force a new type of spray gun simulation
        RDK.Spray_SetState(SPRAY_ON)
        exit()


    # Create a new spray gun object in RoboDK for material deposition (3D printing simulation)
    # by using RDK.Spray_Add(tool, object, options_command, volume, geometry)
    # tool: tool item (TCP) to use
    # object: object to project the particles
    # options_command (optional): string to specify options. Example:
    #     STEP=AxB: Defines the grid to be projected 1x1 means only one line of particle projection (for example, for welding)
    #     PARTICLE: Defines the shape and size of particle (sphere or particle), unless a specific geometry is provided:
    #       a- SPHERE(radius, facets)
    #       b- SPHERE(radius, facets, scalex, scaley, scalez)
    #       b- CUBE(sizex, sizey, sizez)
    #     RAND=factor: Defines a random factor factor 0 means that the particles are not deposited randomly
    #     ELLYPSE: defines the volume as an ellypse (default)
    #     RECTANGLE: defines the volume as a rectangle
    #     PROJECT: project the particles to the surface (default) (for welding, painting or scanning)
    #     NO_PROJECT: does not project the particles to the surface (for example, for 3D printing)
    #
    # volume (optional): Matrix of parameters defining the volume of the spray gun
    # geometry (optional): Matrix of vertices defining the triangles.


    diameter = 22.225 # in mm
    detail = 8 # number of rings of detail to display the sphere
    scale = '1,1,0.5' # scale the particle in 0.5 along the tool Z axis (simulating gravity effect)
    options_command = "ELLYPSE NO_PROJECT PARTICLE=SPHERE(%.3f,%.0f,%s)" % (diameter, detail, scale) # simulate
    #options_command = "PARTICLE=CUBE(10,10,2) STEP=8x8"
    #options_command = "PARTICLE=SPHERE(4,8) STEP=8x8"
    #options_command = "PARTICLE=SPHERE(4,8,1,1,0.1) STEP=8x8 RAND=3"

    # Example commands for welding:
    # options_command = "PROJECT PARTICLE=SPHERE(4,8)"
    # options_command = PARTICLE=SPHERE(4,8) STEP=1x0

    tool = 0    # auto detect active tool
    obj = 0     # auto detect object in active reference frame

    # Material is deposited at 0,0,0 with respect to the TCP coordinates
    close_param = [0,0,0,  0,0,0,  0,0,0,     0.7,0.5,0.8,1] # color as RGBA
    far_param   = [0,0,0,  0,0,0,  0,0,0,     0.7,0.5,0.8,1] # color as RGBA
    volume = Mat([close_param, far_param])
    RDK.Spray_Add(tool, obj, options_command, volume.tr())
    RDK.Spray_SetState(SPRAY_ON)

--- Python program SimulateFinalResult ---
# This script will simulate the final result of the 3D printed part using the Spray function

# Or visit: http://www.robodk.com/doc/PythonAPI/
# Note: you do not need to keep a copy of this file, your python script is saved with the station
from robolink import *    # API to communicate with RoboDK
from robodk import *      # basic matrix operations


RENDER = True      # Set to False
STEP_MM = 2         # Detail step in MM for linear moves
STEP_DEG = 2        # Detail step in DEG for joint moves

# Start a connection with the RoboDK API
RDK = Robolink()

# Select the first/only robot in the cell:
program = RDK.ItemUserPick('Select a program to simulate', ITEM_TYPE_PROGRAM)
if not program.Valid():
    raise Exception("No program available")

# Get the robot
robot = RDK.Item('', ITEM_TYPE_ROBOT)
#robot = program.getLink(ITEM_TYPE_ROBOT) # available in newer versions
if not robot.Valid():
    raise Exception("No robot available")

progname = program.Name()
print("Using program %s" % progname)


# Get the program as a list of joint values
tool = robot.getLink(ITEM_TYPE_TOOL)
progok_jlist = program.InstructionListJoints(STEP_MM, STEP_DEG)
progok = progok_jlist[0] # progok: String that indicates if there are any issues with the program
jlist = progok_jlist[1]  # jlist: list of joints

# Check that the program is correct and has at least a movement
njoints = jlist.size(1)
if njoints < 1:
    raise Exception("Program %s has no movements" % name)

# Check if there are any issues with the program:
if progok != "Success":
    raise Exception("Problems with program %s: %s." %(name, progok))

# Reset any material deposition simulation
RDK.Spray_Clear()

robot.setPoseTool(tool)

# Start material deposition simulation according to the Extruder script
RDK.RunProgram('Extruder(0)')
# Alternatively:
#RDK.Item('Extruder', ITEM_TYPE_PYTHON).RunProgram([1])

if not RENDER:
    RDK.Render(False)

# Iterate through all joints in the matrix and check for collisions
njoints_all = jlist.size(1)
for i in range(njoints_all):
    ji = jlist[:,i].tolist()

    # Update the robot to a new position (it will create a new particle)
    robot.setJoints(ji)
    if not RENDER:
        # If Render is turned off (faster) update the position to draw a new particle
        RDK.Update()

    # Show a message in the RoboDK status bar from time to time
    if i % 10 == 0:
        msg = "Quick material deposition simulation for %s (%.1f %%)" % (progname, 100.0*(i/njoints_all))
        print(msg)
        RDK.ShowMessage(msg, False)

    # Render from time to time even if we have render deactivated
    if not RENDER and i % 500 == 0:
        RDK.Render()

RDK.Render(True)
msg = "Done"
print("Done")
RDK.ShowMessage(msg, False)
